{attribute 'hide_all_locals'}
FUNCTION_BLOCK ResetGroup IMPLEMENTS ITask
VAR_INPUT
END_VAR
VAR_OUTPUT
END_VAR
VAR
	groupReset			: MC_GroupReset;
	_caGroup			: ICollisionGroup;
	State: INT;
	_resetGroup : BOOL;
	_busy : BOOL;
	_error : BOOL;
	_done : BOOL;
END_VAR

CASE State OF
	0:
		IF _resetGroup THEN
			_done := FALSE;
			_error := FALSE;
			_busy := TRUE;
			groupReset.Execute := TRUE;
			IF groupReset.Busy THEN
				State := 10;
				_resetGroup := FALSE;
			END_IF
		END_IF
	
	10:
		IF NOT groupReset.Busy THEN
			IF groupReset.Done THEN
				_done := TRUE;
			ELSIF groupReset.Error THEN
				_error := TRUE;
			END_IF
			_busy := FALSE;
			groupReset.Execute := false;
			State := 0;
		END_IF
END_CASE


groupReset(AxesGroup := _caGroup.GroupRef);

METHOD Abort : BOOL
groupReset.Execute := FALSE;
State := 0;
Abort := true;
END_METHOD

PROPERTY Busy : BOOL
GET
Busy := _busy;
END_GET
END_PROPERTY

PROPERTY Done : BOOL
GET
Done := _done;
END_GET
END_PROPERTY

PROPERTY Error : BOOL
GET
Error := _error;
END_GET
END_PROPERTY

METHOD Execute : BOOL
Execute := _resetGroup := true;
END_METHOD

METHOD FB_init : BOOL
VAR_INPUT
	bInitRetains : BOOL; // if TRUE, the retain variables are initialized (warm start / cold start)
	bInCopyCode : BOOL;  // if TRUE, the instance afterwards gets moved into the copy code (online change)
	CAGroup : ICollisionGroup;	
END_VAR
_caGroup := CAGroup;
END_METHOD

END_FUNCTION_BLOCK

(* stored: Version 1.1.0.1, ProductVersion 3.1.4024.9
   POU ResetGroup: Id {c21d861d-7057-4a32-9917-b2f2f1a5c489}, SpecialFunc None
   Method Abort: Id {6df41d98-0ac8-4a32-bfbe-e6164194489d}
   Property Busy: Id {40717454-2de9-4a99-99e8-2688c5d1093b}
   Get Get: Id {36e751d1-cd0d-4140-9d13-7fc8dd926ebe}
   Property Done: Id {75a96548-58e1-486c-abce-7d1b8fe5bee0}
   Get Get: Id {3f1084b4-4ce2-44c2-8a35-b900f7991a43}
   Property Error: Id {c6c02998-cc81-4d92-a0b0-f7eadd404146}
   Get Get: Id {6dd03e4f-22bd-42a0-ad4c-5237d668c988}
   Method Execute: Id {4246d386-cbbc-455d-868d-690bdbd269ef}
   Method FB_init: Id {56320f66-2e0e-4d3d-8693-c73b3dde8a23} *)
